TYPE ST_EP9224_out :
STRUCT
	stOutput : ARRAY [1..EP9224_NUM_CHANNELS] OF ST_EP9224_OutputChannel;
	bGlobalReset : BOOL;
END_STRUCT
END_TYPE

(* stored: Version 1.1.0.1, ProductVersion 3.1.4024.9
   DUT ST_EP9224_out: Id {1963562e-be7f-42d9-a6c8-cc3d500e693b} *)
